TYPE ST_ControlStewart :
STRUCT
	// Velocity setpint to stewart
	u : ARRAY[0..5] OF LREAL;
	u_t : ARRAY[0..5] OF LREAL;
	
END_STRUCT
END_TYPE

(* stored: Version 1.1.0.1, ProductVersion 3.1.4026.8
   DUT ST_ControlStewart: Id {704a2649-8967-48fa-9ab9-06bf666f146b} *)
